FUNCTION_BLOCK F_MUX_2_1 (* Service Interface Function Block Type *)
  (* Description: Copyright (c) 2012 Profactor GmbH This program and the accompanying materials are made available under the terms of the Eclipse Public License 2.0 which is available at https://www.eclipse.org/legal/epl-2.0/ SPDX-License-Identifier: EPL-2.0 *)
  (* Version 1.0, 2012-05-09, Matthias Plasch, Profactor GmbH *)
  {SET_ATTRIBUTE(GenericClassName, 'GEN_F_MUX')}
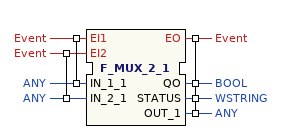
  EVENT_INPUT
    EI1 WITH IN_1_1; (* event input 1 *)
    EI2 WITH IN_2_1; (* event input 2 *)
  END_EVENT
  EVENT_OUTPUT
    EO WITH QO, STATUS, OUT_1; (* merge event output *)
  END_EVENT
  VAR_INPUT
    IN_1_1 : ANY;
    IN_2_1 : ANY;
  END_VAR
  VAR_OUTPUT
    QO : BOOL; (* Event Output Qualifier *)
    STATUS : WSTRING; (* Service Status *)
    OUT_1 : ANY; (* meged data output *)
  END_VAR
  (* Service APPLICATION/RESOURCE: Service Interface Function Block Type *)
END_FUNCTION_BLOCK
